FUNCTION_BLOCK EventLogger
VAR	PERSISTENT
	CurrentEventBufferIndex		: INT:=0;
END_VAR
VAR CONSTANT
	MAX_SIZE_OF_EVENT_BUFFER	: INT:=500;
END_VAR

METHOD PUBLIC AddEvent : BOOL
VAR_INPUT
	What_happend			: STRING[20];
	sEventText				: STRING[255];
	eEventType				: E_EventType;
	eEventSeverity			: TcEventSeverity;
END_VAR
IF NOT isEventBufferFull() THEN
	CurrentEventBufferIndex:=CurrentEventBufferIndex+1;
	GVL.EventBuffer[CurrentEventBufferIndex].eEventType:=eEventType;
	GVL.EventBuffer[CurrentEventBufferIndex].What_happend:=What_happend;
	GVL.EventBuffer[CurrentEventBufferIndex].sEventText:=sEventText;
	GVL.EventBuffer[CurrentEventBufferIndex].eEventSeverity:=eEventSeverity;
	F_UpdateEvent(stEvent:=GVL.EventBuffer[CurrentEventBufferIndex]);
	AddEvent:=TRUE;
ELSE 
	CurrentEventBufferIndex:=0;
END_IF
END_METHOD

METHOD PRIVATE isEventBufferFull : BOOL
VAR_INPUT
END_VAR
IF (CurrentEventBufferIndex+1)>MAX_SIZE_OF_EVENT_BUFFER THEN
	isEventBufferFull:=TRUE;
	ELSE isEventBufferFull:=FALSE;
END_IF
END_METHOD

END_FUNCTION_BLOCK

(* stored: Version 1.1.0.1, ProductVersion 3.1.4024.12
   POU EventLogger: Id {2a670000-1b8d-47c8-867b-df677a6f707e}, SpecialFunc None
   Method AddEvent: Id {f0ccb861-5161-4635-9f82-570737a680db}
   Method isEventBufferFull: Id {42f73c1f-6f32-45af-aa29-e80a7aaf2759} *)
